// TwinCAT 3 PLC project TcGeodetic
// ProgramVersion: 3.1.4023.0
// libraries:
//   Tc2_Standard, * (Beckhoff Automation GmbH)
//   Tc2_System, * (Beckhoff Automation GmbH)
//   Tc3_Module, * (Beckhoff Automation GmbH)
//   TcGeodetic, * (Burks Engineering)
//   TcTransform, * (Burks Engineering)
//   TcUnit, * (www.tcunit.org)
// project tree:
//   / PlcTask.TcTTO
//   TESTs/ FB_GeoPosition_Test.TcPOU, FB_GeoEllipsoid_Test.TcPOU, PRG_TEST.TcPOU
// real-time tasks:
//   TASK PlcTask: cycle T#10ms, priority 20, ADS port 350

CONFIGURATION TcGeodetic
    RESOURCE PLC ON TwinCAT3
        TASK PlcTask(INTERVAL := T#10ms, PRIORITY := 20);
        PROGRAM PRG_TEST WITH PlcTask : PRG_TEST;
    END_RESOURCE
END_CONFIGURATION

// ---- TESTs/PRG_TEST.TcPOU
PROGRAM PRG_TEST
VAR
	fb_GeoPosition : FB_GeoPosition_Test;
	fb_GeoEllipsoid : FB_GeoEllipsoid_Test;
END_VAR

TcUnit.RUN();

END_PROGRAM

// ---- TESTs/FB_GeoPosition_Test.TcPOU
FUNCTION_BLOCK FB_GeoPosition_Test EXTENDS FB_TestSuite
VAR_INPUT
END_VAR
VAR_OUTPUT
END_VAR
VAR
END_VAR

WhenValuesSetExpectValuesRetained();

METHOD PRIVATE WhenValuesSetExpectValuesRetained
VAR_INPUT
	
END_VAR
VAR
	P1 : GeoPosition;
	P1b : GeoPosition;
	P2 : GeoPosition;
	P3 : GeoPosition;
END_VAR
TEST('WhenValuesSetExpectValuesRetained');

// @TEST-RUN
P1.SetFromComponentsRad(PI,PI,1);
P1b.SetFromComponentsRad(PI,PI,1);
P2 := P1;
P3.SetFromComponentsDeg(180,180,1);

// @TEST-ASSERT
AssertTrue(P1.IsEqual(P1b), 'equals check does not work');
AssertTrue(P1.IsEqual(P3),'radians and degrees do not agree');
AssertTrue(P2.LatitudeDeg > 179.99,'latitude not retained');
AssertTrue(P2.LongitudeDeg > 179.99,'longitude not retained');
AssertTrue(P2.Elevation = 1,'elevation not retained');


TEST_FINISHED();
END_METHOD

END_FUNCTION_BLOCK

// ---- TESTs/FB_GeoEllipsoid_Test.TcPOU
FUNCTION_BLOCK FB_GeoEllipsoid_Test EXTENDS FB_TestSuite
VAR_INPUT
END_VAR
VAR_OUTPUT
END_VAR
VAR
END_VAR

WhenReferenceConstantExpectItExists();
WhenGetCartesianExpectValue();
WhenGetGeodeticExpectValue();
WhenTransformEnuAltExpectValue();
WhenTransformEnulatLonExpectValue();

METHOD PRIVATE WhenGetCartesianExpectValue
VAR_INPUT
	
END_VAR
VAR
	PX : GeoPosition;
	PY : GeoPosition;
	PZ : GeoPosition;
	VX : Vector3;
	VY : Vector3;
	VZ : Vector3;
END_VAR
TEST('WhenGetCartesianExpectValue');

// @TEST-RUN
PX.SetFromComponentsDeg(0,0,1);
PY.SetFromComponentsDeg(0,90,1);
PZ.SetFromComponentsDeg(90,0,1);
VX := GeoEllipsoids.WGS84.GetCartesianFromGeodetic(PX);
VY := GeoEllipsoids.WGS84.GetCartesianFromGeodetic(PY);
VZ := GeoEllipsoids.WGS84.GetCartesianFromGeodetic(PZ);

// @TEST-ASSERT
AssertTrue(VX.X = GeoEllipsoids.WGS84.SemiMajorAxis+1, 'X axis check does not work');
AssertTrue(VY.Y = GeoEllipsoids.WGS84.SemiMajorAxis+1, 'Y axis check does not work');
AssertTrue(VZ.Z = (1-GeoEllipsoids.WGS84.Flattening)*GeoEllipsoids.WGS84.SemiMajorAxis +1, 'Z axis check does not work');


TEST_FINISHED();
END_METHOD

METHOD PRIVATE WhenGetGeodeticExpectValue
VAR_INPUT
	
END_VAR
VAR
	PX : GeoPosition;
	PY : GeoPosition;
	PZ : GeoPosition;
	PXYZ : GeoPosition;
	VX : Vector3;
	VXb : Vector3;
	VY : Vector3;
	VZ : Vector3;
	VXYZ : Vector3;
	PX2 : GeoPosition;
	PX2b : GeoPosition;
	PY2 : GeoPosition;
	PZ2 : GeoPosition;
	PXYZ2 : GeoPosition;
END_VAR
TEST('WhenGetGeodeticExpectValue');

// @TEST-RUN
PX.SetFromComponentsDeg(0,0,1);
PY.SetFromComponentsDeg(0,90,1);
PZ.SetFromComponentsDeg(90,0,1);
PXYZ.SetFromComponentsDeg(45,45,1000);
VX := GeoEllipsoids.WGS84.GetCartesianFromGeodetic(PX);
VXb := GeoEllipsoids.WGS84.GetCartesianFromGeodetic(PX);
VXb.Z := VXb.Z - 1;//just south of equator
VY := GeoEllipsoids.WGS84.GetCartesianFromGeodetic(PY);
VZ := GeoEllipsoids.WGS84.GetCartesianFromGeodetic(PZ);
VXYZ := GeoEllipsoids.WGS84.GetCartesianFromGeodetic(PXYZ);
PX2 := GeoEllipsoids.WGS84.GetGeodeticFromCartesian(VX);
PX2b := GeoEllipsoids.WGS84.GetGeodeticFromCartesian(VXb);
PY2 := GeoEllipsoids.WGS84.GetGeodeticFromCartesian(VY);
PZ2 := GeoEllipsoids.WGS84.GetGeodeticFromCartesian(VZ);
PXYZ2 := GeoEllipsoids.WGS84.GetGeodeticFromCartesian(VXYZ);

// @TEST-ASSERT
AssertTrue(PX.IsNearlyEqual(PX2,1E-6,1E-3), 'X axis check does not work');
AssertTrue(PY.IsNearlyEqual(PY2,1E-6,1E-3), 'Y axis check does not work');
AssertTrue(PZ.IsNearlyEqual(PZ2,1E-6,1E-3), 'Z axis check does not work');
AssertTrue(PXYZ.IsNearlyEqual(PXYZ2,1E-6,1E-3), 'Compound axis check does not work');

AssertTrue(PX2b.LatitudeRad < 0, 'Small latitude perturbation does not work');


TEST_FINISHED();
END_METHOD

METHOD PRIVATE WhenReferenceConstantExpectItExists
VAR_INPUT
END_VAR
VAR
	WGS84 : REFERENCE TO GeoEllipsoid;
END_VAR
TEST('WhenReferenceConstantExpectItExists');

// @TEST-RUN
WGS84 REF=  GeoEllipsoids.WGS84;

// @TEST-ASSERT
AssertTrue(WGS84.SemiMajorAxis = 6378137, 'semi major axis not right');
AssertTrue(WGS84.Flattening = 1.0 / 298.257223563, 'flattening not right');

TEST_FINISHED();
END_METHOD

METHOD PRIVATE WhenTransformEnuAltExpectValue
VAR_INPUT
	
END_VAR
VAR
	Psurf : GeoPosition;
	Palt : GeoPosition;
	Vsurf : Vector3;
	Valt : Vector3;
	Valt_surf : Vector3;
	Hsurf : HMatrix;
	Valt2 : Vector3;
END_VAR
TEST('WhenTransformEnuAltExpectValue');

// @TEST-RUN
Psurf.SetFromComponentsDeg(0,0,0);
Palt.SetFromComponentsDeg(PSurf.LatitudeDeg,PSurf.LongitudeDeg,1000);
Valt_surf.SetFromComponents(0,0,Palt.Elevation);

Vsurf := GeoEllipsoids.WGS84.GetCartesianFromGeodetic(Psurf);
Valt := GeoEllipsoids.WGS84.GetCartesianFromGeodetic(Palt);
Hsurf := GeoEllipsoids.WGS84.GetTangentEnuTransform(Psurf);
Valt2 := Hsurf.GetTransformedVector3(Valt_surf);

// @TEST-ASSERT
AssertTrue(Valt.IsNearlyEqual(Valt2,1E-6), 'transformation did not work');


TEST_FINISHED();
END_METHOD

METHOD PRIVATE WhenTransformEnuLatLonExpectValue
VAR_INPUT
	
END_VAR
VAR
	Psurf : GeoPosition;
	Palt : GeoPosition;
	Vsurf : Vector3;
	Valt : Vector3;
	Valt_surf : Vector3;
	Hsurf : HMatrix;
	Valt2 : Vector3;
END_VAR
TEST('WhenTransformEnuLatLonExpectValue');

// @TEST-RUN
Psurf.SetFromComponentsDeg(10,10,0);
Palt.SetFromComponentsDeg(PSurf.LatitudeDeg,PSurf.LongitudeDeg,1000);
Valt_surf.SetFromComponents(0,0,Palt.Elevation);

Vsurf := GeoEllipsoids.WGS84.GetCartesianFromGeodetic(Psurf);
Valt := GeoEllipsoids.WGS84.GetCartesianFromGeodetic(Palt);
Hsurf := GeoEllipsoids.WGS84.GetTangentEnuTransform(Psurf);
Valt2 := Hsurf.GetTransformedVector3(Valt_surf);

// @TEST-ASSERT
AssertTrue(Valt.IsNearlyEqual(Valt2,1E-6), 'transformation did not work');


TEST_FINISHED();
END_METHOD

END_FUNCTION_BLOCK
